FUNCTION_BLOCK FB_ADD
VAR_INPUT
	int1,int2:INT;
END_VAR
VAR_OUTPUT
	out:int;
END_VAR
VAR
END_VAR

out:=int1+int2;

END_FUNCTION_BLOCK

(* stored: Version 1.1.0.1, ProductVersion 3.1.4024.3
   POU FB_ADD: Id {a13bdbc9-ce5c-4839-afa2-9aebe5957e6b}, SpecialFunc None *)
